VAR_GLOBAL
    bReady  : BOOL := TRUE;
    nLimit  : INT := 10;
    rFactor : REAL := 1.0;
    sLabel  : STRING := 'Sample';
END_VAR

(* stored: Version 1.1.0.1, ProductVersion 3.1.4024.10 *)
